// SIMATIC S7-200 project (STEP 7-Micro/WIN), CPU 221 REL 01.10

ORGANIZATION_BLOCK 主:OB1
TITLE=
// 烤箱通过连接热电偶或其他传感器的模拟输入监测温度，并将其转换为摄氏度的数字值，确保温度测量始终准确反映实际环境。温度设定值被预设为一个固定值，以确保控制稳定。PID控制器根据测量温度与设定值之间的差异计算加热元件的必要功率水平，输出控制信号驱动模拟输出调节加热强度。模拟输出的计算方式为16000减去缩放后的PID输出，确保当温度低于设定值时加热功率增加，而当温度过高时功率减少，其值保持在合理范围内以维持控制精度。为了确保安全，当测量温度等于或超过设定值时，加热元件的功率会立即降低到最低水平，通过将模拟输出设为特定值实现，以保护设备和实验。此外，数字输出控制一个冷却风扇，帮助维持烤箱内的最佳条件，风扇在模拟输出相关值较小时开启，较大时关闭，处于中间范围时保持当前状态。
// 
BEGIN
Network 1 // 设置通讯方式，调用传送PID参数子程序，启动TD200使能位。
//  
// 网络注释
//  
// 
LD     SM0.1
MOVB   9, SMB30
MOVB   0, SMB130
CALL   SBR_0:SBR0
MOVB   16#80, VB12
MOVB   0, MB0
?000
Network 2 // 传送向PC机发送的数据表。
// 
// 
LD     SM0.0
MOVB   4, VB199
MOVW   VW56, VW200
MOVW   VW76, VW202
Network 3 // 向PC机发送数据。
// 
// 
LD     SM0.5
EU
XMT    VB199, 0
Network 4 // 超过额温度限制输出。
// 
// 
LDD>=  VD100, VD104
MOVW   +16000, AQW0
Network 5 // 温控时间的计数器（单位为秒）。
// 
// 
LD     SM0.5
LD     SM0.1
CTU    C0, +0
Network 6 // 计算检测的温度参数，传送到VW556。设定的温度参数传送到VW576。
// 
// 
LD     SM0.0
MOVR   VD100, AC0
*R     32000.0, AC0
ROUND  AC0, AC0
DTI    AC0, VW556
MOVR   VD104, AC0
*R     32000.0, AC0
ROUND  AC0, AC0
DTI    AC0, VW576
Network 7 // 检测的温度值送VW56，设定温度值送VW76。
// 
// 
LD     SM0.0
-I     +6552, VW556
MOVW   VW556, VW56
/I     +131, VW56
-I     +6552, VW576
MOVW   VW576, VW76
/I     +131, VW76
END_ORGANIZATION_BLOCK

SUBROUTINE_BLOCK SBR_0:SBR0
TITLE= 
// 子程序注释
// 按 F1 获得帮助及举例程序
//  
// 
BEGIN
Network 1 // 传送PID参数。
//  
// 网络注释
//  
// 
LD     SM0.0
MOVR   0.615, VD104
MOVR   2.0, VD112
MOVR   0.1, VD116
MOVR   4.0, VD120
MOVR   0.0, VD124
MOVB   10, SMB34
ATCH   INT_0:INT0, 10
ENI
END_SUBROUTINE_BLOCK

INTERRUPT_BLOCK INT_0:INT0
TITLE= 
// 中断程序注释
// 按 F1 获得帮助及举例程序
//  
// 
BEGIN
Network 1 // 检测温度参数送PID参数表。
//  
// 网络注释
//  
// 
LD     SM0.5
EU
MOVW   AIW0, VW402
DTR    VD400, VD404
MOVR   VD404, VD408
/R     32000.0, VD408
MOVR   VD408, VD100
Network 2 // I0.0=1,计算PID输出。
// 
// 
LD     I0.0
PID    VB100, 0
Network 3 // 根据PID输出通过D/A模块控制调压模块（DC 0-5V）。
// 
// 
LD     SM0.0
MOVR   VD108, AC0
*R     16000.0, AC0
ROUND  AC0, AC0
DTI    AC0, VW310
MOVW   +16000, VW304
-I     VW310, VW304
MOVW   VW304, AQW0
Network 4 // ****用Q0.0控制交流220V的输出。
// 
// 
LD     SM0.0
LPS
AW>    VW304, +10000
R      Q0.0, 1
LPP
AW<    VW304, +6000
S      Q0.0, 1
END_INTERRUPT_BLOCK
